{attribute 'qualified_only'}
{attribute 'strict'}
TYPE E_PHASING_STATE_MACHINE :
(
	POWER_OFF := 0,
	POWER_ON :=1,
	ACCELERATION :=2,
	PHASING :=3
);
END_TYPE

(* stored: Version 1.1.0.1, ProductVersion 3.1.4022.3
   DUT E_PHASING_STATE_MACHINE: Id {194eca20-5771-4216-89ae-ef0127731437} *)
